// TwinCAT 3 PLC project PRG_MachineSystem
// Title: B_MachineSystem
// Company: RafalOS
// Author: Rafał Osajda
// ProjectVersion: 0.0.0.19
// ProgramVersion: 3.1.4024.0
// libraries:
//   B_Base, * (RafalOS)
//   B_Base_HMI_Connector, * (RafalOS)
//   B_HMIElements, * (RafalOS)
//   B_HMIManager, * (RafałOS)
//   B_IO, * (RafalOS)
//   B_MachineControl, * (RafalOS)
//   B_MachineControl_HMI_Connector, * (RafalOS)
//   B_StatesAndModes, * (RafalOS)
//   Tc2_Standard, * (Beckhoff Automation GmbH)
//   Tc2_System, * (Beckhoff Automation GmbH)
//   Tc3_Module, * (Beckhoff Automation GmbH)
// project tree:
//   GVLs/ GVL_MCSafety.TcGVL, GVL_RequeestChange.TcGVL, GVL_SystemVariable.TcGVL
//   / PlcTask.TcTTO
//   POUsCompilation/ Compilation.TcPOU
//   POUs/01_MachineDefaultConfiguration/ FB_MachineDefaultConfiguration.TcPOU
//   POUs/02_HMIDefaultConfiguration/ FB_DefaultHMIConfiguration.TcPOU
//   POUs/03_CreatingTempleteRecipe/ FB_DefaultTemplate.TcPOU
//   POUs/ PRG_ControlHMI.TcPOU, PRG_ControlHMIInit.TcPOU, PRG_SystemControlMachineInit.TcPOU, PRG_SystemControlMachineWork.TcPOU, ST_MainMenuButton.TcDUT, ST_PrepareDataModules.TcDUT

CONFIGURATION PRG_MachineSystem
    RESOURCE PLC ON TwinCAT3
        TASK PlcTask(INTERVAL := T#10ms, PRIORITY := 20);
        PROGRAM Compilation WITH PlcTask : Compilation;
        PROGRAM PRG_ControlHMI WITH PlcTask : PRG_ControlHMI;
        PROGRAM PRG_SystemControlMachineInit WITH PlcTask : PRG_SystemControlMachineInit;
        PROGRAM PRG_SystemControlMachineWork WITH PlcTask : PRG_SystemControlMachineWork;
        PROGRAM PRG_ControlHMIInit WITH PlcTask : PRG_ControlHMIInit;
    END_RESOURCE
END_CONFIGURATION

// ---- POUs/ST_MainMenuButton.TcDUT
TYPE ST_MainMenuButton :
STRUCT
	fbMMB0_MainScreen			: FB_HMIEButton;
	fbMMB1_Recipe				: FB_HMIEButton;
	fbMMB2_Parameters			: FB_HMIEButton;
	fbMMB3_Events				: FB_HMIEButton;
	fbMMB4_ModeChange			: FB_HMIEButton;
	fbMMB5_Statistics			: FB_HMIEButton;
	fbMMB6_StateDiagram			: FB_HMIEButton;
	fbMMB7_Settings				: FB_HMIEButton;

	fbMMB0_MainScreen_HMI_Connector		: FB_HMIEButton_HMI (itfBaseLoggerConnector := GVL_SystemVariable.fbLogger, itfButton := fbMMB0_MainScreen);
	fbMMB1_Recipe_HMI_Connector			: FB_HMIEButton_HMI (itfBaseLoggerConnector := GVL_SystemVariable.fbLogger, itfButton := fbMMB1_Recipe);
	fbMMB2_Parameters_HMI_Connector		: FB_HMIEButton_HMI (itfBaseLoggerConnector := GVL_SystemVariable.fbLogger, itfButton := fbMMB2_Parameters);
	fbMMB3_Events_HMI_Connector			: FB_HMIEButton_HMI (itfBaseLoggerConnector := GVL_SystemVariable.fbLogger, itfButton := fbMMB3_Events);
	fbMMB4_ModeChange_HMI_Connector		: FB_HMIEButton_HMI (itfBaseLoggerConnector := GVL_SystemVariable.fbLogger, itfButton := fbMMB4_ModeChange);
	fbMMB5_Statistics_HMI_Connector		: FB_HMIEButton_HMI (itfBaseLoggerConnector := GVL_SystemVariable.fbLogger, itfButton := fbMMB5_Statistics);
	fbMMB6_StateDiagram_HMI_Connector	: FB_HMIEButton_HMI (itfBaseLoggerConnector := GVL_SystemVariable.fbLogger, itfButton := fbMMB6_StateDiagram);
	fbMMB7_Settings_HMI_Connector		: FB_HMIEButton_HMI (itfBaseLoggerConnector := GVL_SystemVariable.fbLogger, itfButton := fbMMB7_Settings);
	
END_STRUCT
END_TYPE

// ---- POUs/ST_PrepareDataModules.TcDUT
TYPE ST_PrepareDataModules :
STRUCT
	fbPrepareDataModul_Empty			: FB_MCHMIPrepareDataForScreen;
	fbPrepareDataModul_00_01			: FB_MCHMIPrepareDataForScreen_00_01;
	fbPrepareDataModul_00_02			: FB_MCHMIPrepareDataForScreen_00_02;
	fbPrepareDataModul_00_03			: FB_MCHMIPrepareDataForScreen_00_03;
	fbPrepareDataModul_00_04			: FB_MCHMIPrepareDataForScreen_00_04;
	fbPrepareDataModul_00_05			: FB_MCHMIPrepareDataForScreen_00_05;
	fbPrepareDataModul_01_XX			: FB_MCHMIPrepareDataForScreen_01_XX;	//parametry
	fbPrepareDataModul_02_XX			: FB_MCHMIPrepareDataForScreen_02_XX;	//receptury
	fbPrepareDataModul_03_XX			: FB_MCHMIPrepareDataForScreen_03_XX;	//alarmy 
	fbPrepareDataModul_04_XX			: FB_MCHMIPrepareDataForScreen_04_XX;	//zmiana trybu
	fbPrepareDataModul_05_XX			: FB_MCHMIPrepareDataForScreen_05_XX;	//statystyki
	fbPrepareDataModul_06_XX			: FB_MCHMIPrepareDataForScreen_06_XX;	//diagram
	fbPrepareDataModul_07_XX			: FB_MCHMIPrepareDataForScreen_07_XX;	//ustawienia
END_STRUCT
END_TYPE

// ---- GVLs/GVL_MCSafety.TcGVL
{attribute 'qualified_only'}
VAR_GLOBAL
	flSS1				: FB_BaseFlag;
	flSTO				: FB_BaseFlag;
	
END_VAR

// ---- GVLs/GVL_RequeestChange.TcGVL
{attribute 'qualified_only'}
VAR_GLOBAL
//Przyciski zmaiany stanu	
//	fbprUndefined			: FB_RequestChanges;
	fbprAbort				: FB_MCRequiredChange;
  	fbprClear				: FB_MCRequiredChange;
   	fbprReset				: FB_MCRequiredChange;
   	fbprStart				: FB_MCRequiredChange;
   	fbprStop				: FB_MCRequiredChange;
   	fbprHold				: FB_MCRequiredChange;
   	fbprUnhold				: FB_MCRequiredChange;
   	fbprSuspend				: FB_MCRequiredChange;
   	fbprUnsuspend			: FB_MCRequiredChange;
  	fbprComplete			: FB_MCRequiredChange;
//przyciski zmiany trybu
//	fbprNiedozwolony		: FB_SITP_PolecenieZmianyTrybu (ePolecenie := E_SITP_PolecenieZmianyTrybu.brak);     
	fbprProduction			: FB_MCRequiredChange;
    fbprMaintenance			: FB_MCRequiredChange;
    fbprManual				: FB_MCRequiredChange;
    fbprWashing				: FB_MCRequiredChange;
    fbprDiagnostics			: FB_MCRequiredChange;
//    fbprUzytkownika2		: FB_RequestChanges;
//   fbprUzytkownika3		: FB_RequestChanges;
//    fbprUzytkownika4		: FB_RequestChanges;
//    fbprUzytkownika5		: FB_RequestChanges;

END_VAR

// ---- GVLs/GVL_SystemVariable.TcGVL
{attribute 'qualified_only'}
VAR_GLOBAL
	fbTime							: FB_BaseTime;
	fbLocation						: FB_BaseLocation;
	fbLogger						: FB_BaseLogger;
	stCommonData					: ST_BaseCommonData;
	
	(*	Element FB_MachineControl - sterowanie stanami i trybami pracy	*)
	fbSaMController					: FB_SaMController;
	
	(*	Główny element sterujący maszyną - logika pracy					*)
	fbMachineControl				: FB_MCMachineControl;
	
	(*	Zmienne zakończenia konfiguracji	*)
	bDefaultInitDone				: BOOL;
	bMachineInitDone				: BOOL;
	bControlHMIInit					: BOOL;
	
	(*	receptury	*)
	fbRecipe						: FB_BaseRecipe;
	
END_VAR

// ---- POUsCompilation/Compilation.TcPOU
PROGRAM Compilation
VAR
	fbMachineConfiguration	: FB_MachineDefaultConfiguration;
	fbHMIConfiguration		: FB_DefaultHMIConfiguration;
END_VAR

END_PROGRAM

// ---- POUs/01_MachineDefaultConfiguration/FB_MachineDefaultConfiguration.TcPOU
(*			
	RafalOS
	Rafał Osajda		10.11.2025		TC 4024.66
	Główny blok konfiguracyjny MachineControl
*)
FUNCTION_BLOCK FB_MachineDefaultConfiguration EXTENDS FB_Base IMPLEMENTS ITF_MCConfiguration
VAR

END_VAR

(*			
	RafalOS
	Rafał Osajda		26.11.2025		TC 4024.66
	Dodawanie szablonu receptury
*)
METHOD AddCreateTemplate : BOOL
VAR_INPUT
	itfMachineControl	: B_MachineControl.ITF_MCMachineControlConfigure;
END_VAR
//itfMachineControl.AddCreateTemplateFromConfiguration (fbCreateTemplate := );
END_METHOD

(*			
	RafalOS
	Rafał Osajda		13.11.2025		TC 4024.66
	Metoda przeznaczona do dodawania elementów do FB_MachineControl
*)
METHOD AddElements : BOOL
VAR_INPUT
	itfMachineControl	: B_MachineControl.ITF_MCMachineControlConfigure;
END_VAR
END_METHOD

(*			
	RafalOS
	Rafał Osajda		13.11.2025		TC 4024.66
	Podpięcie menadżera HMI
*)
METHOD AddHMIManager : BOOL
VAR_INPUT
	itfMachineControl	: B_MachineControl.ITF_MCMachineControlConfigure;
END_VAR
itfMachineControl.AddHMIManagerFromConfiguration (fbHMIManager := PRG_ControlHMI.fbHMIManager);
END_METHOD

(*			
	RafalOS
	Rafał Osajda		13.11.2025		TC 4024.66
	Dodanie samego siebie do systemu controli maszyny
*)
METHOD AddMachineCotrolToYourSelf : BOOL
VAR_INPUT
	itfMachineControl			: ITF_MCMachineControlConfigure;
END_VAR
itfMachineControl.AddMachineCotrolToYourSelfFromConfiguration ();
END_METHOD

(*			
	RafalOS
	Rafał Osajda		26.11.2025		TC 4024.66
	Dodanie obsługi receptur
*)
METHOD AddModulRecipe : BOOL
VAR_INPUT
	itfMachineControl	: B_MachineControl.ITF_MCMachineControlConfigure;
END_VAR
itfMachineControl.AddModulRecipeFromConfiguration (itfRecipe := GVL_SystemVariable.fbRecipe);
END_METHOD

(*			
	RafalOS
	Rafał Osajda		13.11.2025		TC 4024.66
	Dodanie modułu sterowania stanami i trybami do machinecontrol
*)
METHOD PUBLIC AddSaMCotrollerToMachineControl : BOOL
VAR_INPUT
	itfMachineControl			: ITF_MCMachineControlConfigure;
END_VAR
itfMachineControl.AddSaMCotrollerToMachineControlFromConfiguration (itfSaMController := GVL_SystemVariable.fbSaMController);
END_METHOD

METHOD AddSaMToTopElement
VAR_INPUT
	itfMachineControl	: B_MachineControl.ITF_MCMachineControlConfigure;
END_VAR
itfMachineControl.AddSaMToTopElementFromConfiguration (itfSaMController := GVL_SystemVariable.fbSaMController);
END_METHOD

(*			
	RafalOS
	Rafał Osajda		13.11.2025		TC 4024.66
	Zlinkowanie danych wspólnych do dodanych elementów
*)
METHOD LinkCommonDataToAddedElements : BOOL
VAR_INPUT
	itfMachineControl	: B_MachineControl.ITF_MCMachineControlConfigure;
END_VAR
itfMachineControl.LinkCommonDataToAddedElementsFromConfiguration (stCommonData := GVL_SystemVariable.stCommonData);
END_METHOD

(*			
	RafalOS
	Rafał Osajda		13.11.2025		TC 4024.66
	Dodanie głównego komunikatora pomiędzy topelementami do topelementów
*)
METHOD LinkMassangerToaddedTopElements : BOOL
VAR_INPUT
	itfMachineControl	: B_MachineControl.ITF_MCMachineControlConfigure;
END_VAR
itfMachineControl.LinkMassangerToaddedTopElementsFromConfiguration (
	fbCommunicator := GVL_SystemVariable.fbMachineControl.GetCommunicatorITF ()
);
END_METHOD

(*			
	RafalOS
	Rafał Osajda		14.11.2025		TC 4024.66
	Podpięcie przyciskow zmiany trybu i stanu
*)
METHOD LinkRequestButtonChange : BOOL
VAR_INPUT
	itfMachineControl	: B_MachineControl.ITF_MCMachineControlConfigure;
END_VAR
itfMachineControl.LinkRequestButtonStateChangeFromConfiguration (iNumberOfRequest := E_SaMCommandChangeState.Clear,		itfRequest := GVL_RequeestChange.fbprClear);
itfMachineControl.LinkRequestButtonStateChangeFromConfiguration (iNumberOfRequest := E_SaMCommandChangeState.Reset, 	itfRequest := GVL_RequeestChange.fbprReset);
itfMachineControl.LinkRequestButtonStateChangeFromConfiguration (iNumberOfRequest := E_SaMCommandChangeState.Start, 	itfRequest := GVL_RequeestChange.fbprStart);
itfMachineControl.LinkRequestButtonStateChangeFromConfiguration (iNumberOfRequest := E_SaMCommandChangeState.Stop, 		itfRequest := GVL_RequeestChange.fbprStop);
itfMachineControl.LinkRequestButtonStateChangeFromConfiguration (iNumberOfRequest := E_SaMCommandChangeState.Suspend, 	itfRequest := GVL_RequeestChange.fbprSuspend);
itfMachineControl.LinkRequestButtonStateChangeFromConfiguration (iNumberOfRequest := E_SaMCommandChangeState.Unsuspend, itfRequest := GVL_RequeestChange.fbprUnsuspend);
itfMachineControl.LinkRequestButtonStateChangeFromConfiguration (iNumberOfRequest := E_SaMCommandChangeState.Hold, 		itfRequest := GVL_RequeestChange.fbprHold);
itfMachineControl.LinkRequestButtonStateChangeFromConfiguration (iNumberOfRequest := E_SaMCommandChangeState.Unhold, 	itfRequest := GVL_RequeestChange.fbprUnhold);
itfMachineControl.LinkRequestButtonStateChangeFromConfiguration (iNumberOfRequest := E_SaMCommandChangeState.Complete, 	itfRequest := GVL_RequeestChange.fbprComplete);
itfMachineControl.LinkRequestButtonStateChangeFromConfiguration (iNumberOfRequest := E_SaMCommandChangeState.Abort,		itfRequest := GVL_RequeestChange.fbprAbort);

itfMachineControl.LinkRequestButtonModeChangeFromConfiguration (iNumberOfRequest := E_SaMCommandChangeMode.Production, 	itfRequest := GVL_RequeestChange.fbprProduction);
itfMachineControl.LinkRequestButtonModeChangeFromConfiguration (iNumberOfRequest := E_SaMCommandChangeMode.Maintenance,	itfRequest := GVL_RequeestChange.fbprMaintenance);
itfMachineControl.LinkRequestButtonModeChangeFromConfiguration (iNumberOfRequest := E_SaMCommandChangeMode.Manual, 		itfRequest := GVL_RequeestChange.fbprManual);
itfMachineControl.LinkRequestButtonModeChangeFromConfiguration (iNumberOfRequest := E_SaMCommandChangeMode.Washing,		itfRequest := GVL_RequeestChange.fbprWashing);
itfMachineControl.LinkRequestButtonModeChangeFromConfiguration (iNumberOfRequest := E_SaMCommandChangeMode.Diagnostisc,	itfRequest := GVL_RequeestChange.fbprDiagnostics);
END_METHOD

(*			
	RafalOS
	Rafał Osajda		13.11.2025		TC 4024.66
	Podłączenie wsyzstkich zmiennych pochodzących od Programu safety 
*)
METHOD LinkSafetyToaddedElements : BOOL
VAR_INPUT
	itfMachineControl	: B_MachineControl.ITF_MCMachineControlConfigure;
END_VAR
itfMachineControl.LinkSafetyToaddedElementsFromConfiguration (
	flSS1 := GVL_MCSafety.flSS1,
	flSTO := GVL_MCSafety.flSTO
);
END_METHOD

(*			
	RafalOS
	Rafał Osajda		13.11.2025		TC 4024.66
	Nadanie unikalnych kodów elementom w systemie
*)
METHOD SetCodeToAddedElements : BOOL
VAR_INPUT
	itfMachineControl	: B_MachineControl.ITF_MCMachineControlConfigure;
END_VAR
itfMachineControl.SetCodeToAddedElementsFromConfiguration ();
END_METHOD

(*			
	RafalOS
	Rafał Osajda		13.11.2025		TC 4024.66
	Uruchomienie lub wyłączenie obsługi HMI jak jest false fb obsługi nie jest dodawane do MachineControl
*)
METHOD SetEnableHMIService : BOOL
VAR_INPUT
	itfMachineControl	: B_MachineControl.ITF_MCMachineControlConfigure;
END_VAR
itfMachineControl.SetEnableHMIServiceFromConfiguration (bValue := TRUE);
END_METHOD

(*			
	RafalOS
	Rafał Osajda		13.11.2025		TC 4024.66
	Nadaje unikalne ID zgłoszeniom dodanym do elementów w sesyemie
*)
METHOD SetIDEventsToAddedElements : BOOL
VAR_INPUT
	itfMachineControl	: B_MachineControl.ITF_MCMachineControlConfigure;
END_VAR
itfMachineControl.SetIDEventsToAddedElementsFromConfiguration ();
END_METHOD

(*			
	RafalOS
	Rafał Osajda		13.11.2025		TC 4024.66
	Dodanie wszystkim elementom w systemie unikalnego ID
*)
METHOD SetIDToAddedElements : BOOL
VAR_INPUT
	itfMachineControl	: B_MachineControl.ITF_MCMachineControlConfigure;
END_VAR
itfMachineControl.SetIDToAddedElementsFromConfiguration ();
END_METHOD

(*			
	RafalOS
	Rafał Osajda		14.11.2025		TC 4024.66
	ustawienie trybu poczatkowego
*)
METHOD SetStartMode : BOOL
VAR_INPUT
	itfMachineControl	: B_MachineControl.ITF_MCMachineControlConfigure;
END_VAR
itfMachineControl.SetStartModeFromConfiguration (eStartMode := E_BaseMachineMode.Production);
END_METHOD

METHOD PUBLIC STARE_AddHMIToMachineControl : BOOL
VAR_INPUT
	itfMachineControl			: ITF_MCMachineControlConfigure;
END_VAR
//itfMachineControl.AddHMIManager (itfHMIManager := GVL_SystemVariable.fbHMIManager);
END_METHOD

METHOD PUBLIC STARE_AddTopElementToLogger : BOOL
VAR_INPUT
END_VAR
//GVL_SystemVariable.fbMachineControl.JoinTheLogger ();
END_METHOD

(*			
	RafalOS
	Rafał Osajda		29.10.2025		TC 4024.66
	Dodawanie TopElementu do systemu
*)
METHOD PUBLIC STARE_AddTopElementToMachineControl : BOOL
VAR_INPUT
	itfMachineControl			: ITF_MCMachineControlConfigure;
END_VAR
//THIS^.SetText (eLocation := E_BaseLocation.pl, wsDescription := "System");
//THIS^.SetText (eLocation := E_BaseLocation.en, wsDescription := "System");
//THIS^.SetText (eLocation := E_BaseLocation.de, wsDescription := "System");
//GVL_SystemVariable.fbMachineControl.SetName (stName := THIS^.GetTexts ());
//itfMachineControl.AddTopElementFromConfiguration (fbTopElement	:= GVL_SystemVariable.fbMachineControl);
END_METHOD

METHOD STARE_StateAndModes : BOOL
VAR_INPUT
	itfMachineControl			: ITF_MCMachineControlConfigure;
END_VAR
//itfMachineControl.AddRequestStateChange (iNumberOfRequest := E_SaMCommandChangeState.Clear,		itfRequest := GVL_RequeestChange.fbprClear);
//itfMachineControl.AddRequestStateChange (iNumberOfRequest := E_SaMCommandChangeState.Reset, 	itfRequest := GVL_RequeestChange.fbprReset);
//itfMachineControl.AddRequestStateChange (iNumberOfRequest := E_SaMCommandChangeState.Start, 	itfRequest := GVL_RequeestChange.fbprStart);
//itfMachineControl.AddRequestStateChange (iNumberOfRequest := E_SaMCommandChangeState.Stop, 		itfRequest := GVL_RequeestChange.fbprStop);
//itfMachineControl.AddRequestStateChange (iNumberOfRequest := E_SaMCommandChangeState.Suspend, 	itfRequest := GVL_RequeestChange.fbprSuspend);
//itfMachineControl.AddRequestStateChange (iNumberOfRequest := E_SaMCommandChangeState.Unsuspend, itfRequest := GVL_RequeestChange.fbprUnsuspend);
//itfMachineControl.AddRequestStateChange (iNumberOfRequest := E_SaMCommandChangeState.Hold, 		itfRequest := GVL_RequeestChange.fbprHold);
//itfMachineControl.AddRequestStateChange (iNumberOfRequest := E_SaMCommandChangeState.Unhold, 	itfRequest := GVL_RequeestChange.fbprUnhold);
//itfMachineControl.AddRequestStateChange (iNumberOfRequest := E_SaMCommandChangeState.Complete, 	itfRequest := GVL_RequeestChange.fbprComplete);
//itfMachineControl.AddRequestStateChange (iNumberOfRequest := E_SaMCommandChangeState.Abort,		itfRequest := GVL_RequeestChange.fbprAbort);
//
//itfMachineControl.AddRequestModeChange (iNumberOfRequest := E_SaMCommandChangeMode.Production, 	itfRequest := GVL_RequeestChange.fbprProduction);
//itfMachineControl.AddRequestModeChange (iNumberOfRequest := E_SaMCommandChangeMode.Maintenance,	itfRequest := GVL_RequeestChange.fbprMaintenance);
//itfMachineControl.AddRequestModeChange (iNumberOfRequest := E_SaMCommandChangeMode.Manual, 		itfRequest := GVL_RequeestChange.fbprManual);
//itfMachineControl.AddRequestModeChange (iNumberOfRequest := E_SaMCommandChangeMode.Washing,		itfRequest := GVL_RequeestChange.fbprWashing);
//itfMachineControl.AddRequestModeChange (iNumberOfRequest := E_SaMCommandChangeMode.Diagnostisc,	itfRequest := GVL_RequeestChange.fbprDiagnostics);
END_METHOD

END_FUNCTION_BLOCK

// ---- POUs/PRG_ControlHMI.TcPOU
(*			
	RafalOS
	Rafał Osajda		10.11.2025		TC 4024.66
	Program sterowanie HMI
*)
PROGRAM PRG_ControlHMI
VAR
	(*	Domyślna struktura danych dla HMI	*)
	stHMIData					: ST_HMIManager;
	(*	Główny element sterowania wyświetlaniem na HMI					*)
	fbHMIManager				: FB_HMIManager;
	(*	Domyślne przyciski menu głównego - Logika i łaczniki do HMI	*)
	stMainMenuButton			: ST_MainMenuButton;
	(*	Menu główne - Logika 	*)
	fbMainMenu					: FB_HMIEMenu;
	(*	Menu główne - Łącznik	*)
	fbMainMenu_HMI_Connector	: FB_HMIEMenu_HMI (itfBaseLoggerConnector := GVL_SystemVariable.fbLogger, itfMenu := fbMainMenu);
	(*	Łącznik do Machine Control	*)
	fbMachineControl_HMI_Connector		: FB_MCHMIMachineControl_HMI (itfBaseLoggerConnector := GVL_SystemVariable.fbLogger, itfMachineControlConnector := GVL_SystemVariable.fbMachineControl);
	(*	Moduły przygotowyania danych dla stron	*)
	stPrepareDataModules		: ST_PrepareDataModules;
	(*	Łącznik do receptur		*)
	fbRecipeModul_HMI_Connector	: FB_BaseRecipe_HMI (fbBaseRecipe := GVL_SystemVariable.fbRecipe);
END_VAR


	(*	Wywołanie metody sterowania HMI	*)

IF (GVL_Systemvariable.bDefaultInitDone AND
	GVL_Systemvariable.bMachineInitDone AND
	GVL_SystemVariable.bControlHMIInit AND
	GVL_SystemVariable.fbMachineControl.IsInitDone ()) THEN
	
	fbHMIManager ();
END_IF

END_PROGRAM

// ---- POUs/02_HMIDefaultConfiguration/FB_DefaultHMIConfiguration.TcPOU
(*			
	RafalOS
	Rafał Osajda		10.11.2025		TC 4024.66
	Główny blok konfigurujący HMI
*)
FUNCTION_BLOCK FB_DefaultHMIConfiguration EXTENDS FB_Base IMPLEMENTS ITF_HMIConfiguration
VAR
END_VAR

(*			
	RafalOS
	Rafał Osajda		07.12.2025		TC 4024.66
	Dodawanie elementów do systemmu wyświetlania
*)
METHOD AddElement
VAR_INPUT
	itfHMIManager	: B_HMI_Manager.ITF_HMIManagerConfigure;
END_VAR
END_METHOD

(*			
	RafalOS
	Rafał Osajda		20.11.2025		TC 4024.66
	Dodawanie rozszerzonego wyświetlania danych inna prezenacja danych niż domyślna lista
*)
METHOD AddExtendedDisplayToPrepScrModule : BOOL
VAR_INPUT
	itfHMIManager	: B_HMI_Manager.ITF_HMIManagerConfigure;
END_VAR
//przykład jak rozszerzać w progframie maszyny 
//itfHMIManager.AddExtendedDisplayToPrepScrModuleFromConfiguration (
//	itfModule 		:= PRG_ControlHMI.fbPrepareDataModul_02_XX,
//	itfExtension 	:= PRG_ControlHMI.fbxxxx
//);
END_METHOD

(*			
	RafalOS
	Rafał Osajda		19.11.2025		TC 4024.66
	Dodanie połączenia do MachineControl
*)
METHOD AddMachineControlConnector : BOOL
VAR_INPUT
	itfHMIManager	: B_HMI_Manager.ITF_HMIManagerConfigure;
END_VAR
itfHMIManager.AddMachineControlConnectorFromConfiguration (
	itfMachineControl := PRG_ControlHMI.fbMachineControl_HMI_Connector
);
END_METHOD

(*			
	RafalOS
	Rafał Osajda		14.11.2025		TC 4024.66
	Dodanie do systemu menu głównego 
*)
METHOD AddMainMenu : BOOL
VAR_INPUT
	itfHMIManager	: B_HMI_Manager.ITF_HMIManagerConfigure;
END_VAR
	(*	Utowrzenie menu głównego	*)
THIS^.SetText (eLocation := E_BaseLocation.pl, wsDescription := "Okno główne");
THIS^.SetText (eLocation := E_BaseLocation.en, wsDescription := "Main screen");
THIS^.SetText (eLocation := E_BaseLocation.de, wsDescription := "Hauptbildschirm");
PRG_ControlHMI.stMainMenuButton.fbMMB0_MainScreen.SetName (stName := THIS^.GetTexts ());
PRG_ControlHMI.fbMainMenu.AddButton (fbButton :=PRG_ControlHMI.stMainMenuButton.fbMMB0_MainScreen);
THIS^.SetText (eLocation := E_BaseLocation.pl, wsDescription := "Receptury");
THIS^.SetText (eLocation := E_BaseLocation.en, wsDescription := "Recipe");
THIS^.SetText (eLocation := E_BaseLocation.de, wsDescription := "Rezept");
PRG_ControlHMI.stMainMenuButton.fbMMB1_Recipe.SetName (stName := THIS^.GetTexts ());
PRG_ControlHMI.fbMainMenu.AddButton (fbButton :=PRG_ControlHMI.stMainMenuButton.fbMMB1_Recipe);
THIS^.SetText (eLocation := E_BaseLocation.pl, wsDescription := "Parametry");
THIS^.SetText (eLocation := E_BaseLocation.en, wsDescription := "Parameters");
THIS^.SetText (eLocation := E_BaseLocation.de, wsDescription := "Parameter");
PRG_ControlHMI.stMainMenuButton.fbMMB2_Parameters.SetName (stName := THIS^.GetTexts ());
PRG_ControlHMI.fbMainMenu.AddButton (fbButton :=PRG_ControlHMI.stMainMenuButton.fbMMB2_Parameters);
THIS^.SetText (eLocation := E_BaseLocation.pl, wsDescription := "Zdarzenia");
THIS^.SetText (eLocation := E_BaseLocation.en, wsDescription := "Events");
THIS^.SetText (eLocation := E_BaseLocation.de, wsDescription := "Veranstaltungen");
PRG_ControlHMI.stMainMenuButton.fbMMB3_Events.SetName (stName := THIS^.GetTexts ());
PRG_ControlHMI.fbMainMenu.AddButton (fbButton :=PRG_ControlHMI.stMainMenuButton.fbMMB3_Events);
THIS^.SetText (eLocation := E_BaseLocation.pl, wsDescription := "Zmiana trybu");
THIS^.SetText (eLocation := E_BaseLocation.en, wsDescription := "Mode change");
THIS^.SetText (eLocation := E_BaseLocation.de, wsDescription := "Modusänderung");
PRG_ControlHMI.stMainMenuButton.fbMMB4_ModeChange.SetName (stName := THIS^.GetTexts ());
PRG_ControlHMI.fbMainMenu.AddButton (fbButton :=PRG_ControlHMI.stMainMenuButton.fbMMB4_ModeChange);
THIS^.SetText (eLocation := E_BaseLocation.pl, wsDescription := "Statystyki");
THIS^.SetText (eLocation := E_BaseLocation.en, wsDescription := "Statistics");
THIS^.SetText (eLocation := E_BaseLocation.de, wsDescription := "Statistiken");
PRG_ControlHMI.stMainMenuButton.fbMMB5_Statistics.SetName (stName := THIS^.GetTexts ());
PRG_ControlHMI.fbMainMenu.AddButton (fbButton :=PRG_ControlHMI.stMainMenuButton.fbMMB5_Statistics);
THIS^.SetText (eLocation := E_BaseLocation.pl, wsDescription := "Diagram stanów");
THIS^.SetText (eLocation := E_BaseLocation.en, wsDescription := "State diagram");
THIS^.SetText (eLocation := E_BaseLocation.de, wsDescription := "Zustandsdiagramm");
PRG_ControlHMI.stMainMenuButton.fbMMB6_StateDiagram.SetName (stName := THIS^.GetTexts ());
PRG_ControlHMI.fbMainMenu.AddButton (fbButton :=PRG_ControlHMI.stMainMenuButton.fbMMB6_StateDiagram);
THIS^.SetText (eLocation := E_BaseLocation.pl, wsDescription := "Ustawienia");
THIS^.SetText (eLocation := E_BaseLocation.en, wsDescription := "Settings");
THIS^.SetText (eLocation := E_BaseLocation.de, wsDescription := "Einstellungen");
PRG_ControlHMI.stMainMenuButton.fbMMB7_Settings.SetName (stName := THIS^.GetTexts ());
PRG_ControlHMI.fbMainMenu.AddButton (fbButton :=PRG_ControlHMI.stMainMenuButton.fbMMB7_Settings);
//
PRG_ControlHMI.fbMainMenu_HMI_Connector.AddButton (fbButtonHMI := PRG_ControlHMI.stMainMenuButton.fbMMB0_MainScreen_HMI_Connector);
PRG_ControlHMI.fbMainMenu_HMI_Connector.AddButton (fbButtonHMI := PRG_ControlHMI.stMainMenuButton.fbMMB1_Recipe_HMI_Connector);
PRG_ControlHMI.fbMainMenu_HMI_Connector.AddButton (fbButtonHMI := PRG_ControlHMI.stMainMenuButton.fbMMB2_Parameters_HMI_Connector);
PRG_ControlHMI.fbMainMenu_HMI_Connector.AddButton (fbButtonHMI := PRG_ControlHMI.stMainMenuButton.fbMMB3_Events_HMI_Connector);
PRG_ControlHMI.fbMainMenu_HMI_Connector.AddButton (fbButtonHMI := PRG_ControlHMI.stMainMenuButton.fbMMB4_ModeChange_HMI_Connector);
PRG_ControlHMI.fbMainMenu_HMI_Connector.AddButton (fbButtonHMI := PRG_ControlHMI.stMainMenuButton.fbMMB5_Statistics_HMI_Connector);
PRG_ControlHMI.fbMainMenu_HMI_Connector.AddButton (fbButtonHMI := PRG_ControlHMI.stMainMenuButton.fbMMB6_StateDiagram_HMI_Connector);
PRG_ControlHMI.fbMainMenu_HMI_Connector.AddButton (fbButtonHMI := PRG_ControlHMI.stMainMenuButton.fbMMB7_Settings_HMI_Connector);

itfHMIManager.AddMainMenuFromConfiguration (
	fbMenu := PRG_ControlHMI.fbMainMenu,
	fbMenu_HMI := PRG_ControlHMI.fbMainMenu_HMI_Connector
);
END_METHOD

(*			
	RafalOS
	Rafał Osajda		19.11.2025		TC 4024.66
	Dodanie modułów do przygotowywania stron do wyświetlenia
*)
METHOD AddPrepareScreenModule : BOOL
VAR_INPUT
	itfHMIManager	: B_HMI_Manager.ITF_HMIManagerConfigure;
END_VAR
VAR
	iforScreen	: INT;
	iforMode	: INT;
END_VAR
	(*	Dodanie modułów do machine controil	*)
itfHMIManager.AddPrepareScreenModuleFromConfiguration (itfModule := PRG_ControlHMI.stPrepareDataModules.fbPrepareDataModul_Empty);
itfHMIManager.AddPrepareScreenModuleFromConfiguration (itfModule := PRG_ControlHMI.stPrepareDataModules.fbPrepareDataModul_00_01);
itfHMIManager.AddPrepareScreenModuleFromConfiguration (itfModule := PRG_ControlHMI.stPrepareDataModules.fbPrepareDataModul_00_02);
itfHMIManager.AddPrepareScreenModuleFromConfiguration (itfModule := PRG_ControlHMI.stPrepareDataModules.fbPrepareDataModul_00_03);
itfHMIManager.AddPrepareScreenModuleFromConfiguration (itfModule := PRG_ControlHMI.stPrepareDataModules.fbPrepareDataModul_00_04);
itfHMIManager.AddPrepareScreenModuleFromConfiguration (itfModule := PRG_ControlHMI.stPrepareDataModules.fbPrepareDataModul_00_05);
itfHMIManager.AddPrepareScreenModuleFromConfiguration (itfModule := PRG_ControlHMI.stPrepareDataModules.fbPrepareDataModul_01_XX);
itfHMIManager.AddPrepareScreenModuleFromConfiguration (itfModule := PRG_ControlHMI.stPrepareDataModules.fbPrepareDataModul_02_XX);
itfHMIManager.AddPrepareScreenModuleFromConfiguration (itfModule := PRG_ControlHMI.stPrepareDataModules.fbPrepareDataModul_03_XX);
itfHMIManager.AddPrepareScreenModuleFromConfiguration (itfModule := PRG_ControlHMI.stPrepareDataModules.fbPrepareDataModul_04_XX);
itfHMIManager.AddPrepareScreenModuleFromConfiguration (itfModule := PRG_ControlHMI.stPrepareDataModules.fbPrepareDataModul_05_XX);
itfHMIManager.AddPrepareScreenModuleFromConfiguration (itfModule := PRG_ControlHMI.stPrepareDataModules.fbPrepareDataModul_06_XX);
itfHMIManager.AddPrepareScreenModuleFromConfiguration (itfModule := PRG_ControlHMI.stPrepareDataModules.fbPrepareDataModul_07_XX);


	(*	Przypisanie do wszystkich pól pustego FB *)
FOR iforScreen := 0 TO GVL_HMIEConstans.MAX_NUMBER_OF_BUTTON_IN_MENU DO 
	FOR iforMode := 0 TO GVL_SaMConstans.NUMBER_OF_MODES DO 
		itfHMIManager.LinkPrepareScreenToArrayFromConfiguration (
			iScreen 	:= iforScreen, 
			iMode 		:= iforMode, 
			itfModule 	:= PRG_ControlHMI.stPrepareDataModules.fbPrepareDataModul_Empty
		);
	END_FOR
END_FOR

PRG_ControlHMI.stPrepareDataModules.fbPrepareDataModul_00_01.LinkMachineControlHMI (fbMachineControlHMI := PRG_ControlHMI.fbMachineControl_HMI_Connector);
PRG_ControlHMI.stPrepareDataModules.fbPrepareDataModul_00_02.LinkMachineControlHMI (fbMachineControlHMI := PRG_ControlHMI.fbMachineControl_HMI_Connector);
PRG_ControlHMI.stPrepareDataModules.fbPrepareDataModul_00_03.LinkMachineControlHMI (fbMachineControlHMI := PRG_ControlHMI.fbMachineControl_HMI_Connector);
PRG_ControlHMI.stPrepareDataModules.fbPrepareDataModul_00_04.LinkMachineControlHMI (fbMachineControlHMI := PRG_ControlHMI.fbMachineControl_HMI_Connector);
PRG_ControlHMI.stPrepareDataModules.fbPrepareDataModul_00_05.LinkMachineControlHMI (fbMachineControlHMI := PRG_ControlHMI.fbMachineControl_HMI_Connector);
PRG_ControlHMI.stPrepareDataModules.fbPrepareDataModul_01_XX.LinkMachineControlHMI (fbMachineControlHMI := PRG_ControlHMI.fbMachineControl_HMI_Connector);
PRG_ControlHMI.stPrepareDataModules.fbPrepareDataModul_02_XX.LinkMachineControlHMI (fbMachineControlHMI := PRG_ControlHMI.fbMachineControl_HMI_Connector);
PRG_ControlHMI.stPrepareDataModules.fbPrepareDataModul_03_XX.LinkMachineControlHMI (fbMachineControlHMI := PRG_ControlHMI.fbMachineControl_HMI_Connector);
PRG_ControlHMI.stPrepareDataModules.fbPrepareDataModul_04_XX.LinkMachineControlHMI (fbMachineControlHMI := PRG_ControlHMI.fbMachineControl_HMI_Connector);
PRG_ControlHMI.stPrepareDataModules.fbPrepareDataModul_05_XX.LinkMachineControlHMI (fbMachineControlHMI := PRG_ControlHMI.fbMachineControl_HMI_Connector);
PRG_ControlHMI.stPrepareDataModules.fbPrepareDataModul_06_XX.LinkMachineControlHMI (fbMachineControlHMI := PRG_ControlHMI.fbMachineControl_HMI_Connector);
PRG_ControlHMI.stPrepareDataModules.fbPrepareDataModul_07_XX.LinkMachineControlHMI (fbMachineControlHMI := PRG_ControlHMI.fbMachineControl_HMI_Connector);

	(*	Przypisanie modułów do aktywnych akien 	*)
itfHMIManager.LinkPrepareScreenToArrayFromConfiguration (iScreen := 0, iMode := 1, itfModule := PRG_ControlHMI.stPrepareDataModules.fbPrepareDataModul_00_01);
itfHMIManager.LinkPrepareScreenToArrayFromConfiguration (iScreen := 0, iMode := 2, itfModule := PRG_ControlHMI.stPrepareDataModules.fbPrepareDataModul_00_02);
itfHMIManager.LinkPrepareScreenToArrayFromConfiguration (iScreen := 0, iMode := 3, itfModule := PRG_ControlHMI.stPrepareDataModules.fbPrepareDataModul_00_03);
itfHMIManager.LinkPrepareScreenToArrayFromConfiguration (iScreen := 0, iMode := 4, itfModule := PRG_ControlHMI.stPrepareDataModules.fbPrepareDataModul_00_04);
itfHMIManager.LinkPrepareScreenToArrayFromConfiguration (iScreen := 0, iMode := 5, itfModule := PRG_ControlHMI.stPrepareDataModules.fbPrepareDataModul_00_05);

itfHMIManager.LinkPrepareScreenToArrayFromConfiguration (iScreen := 1, iMode := 1, itfModule := PRG_ControlHMI.stPrepareDataModules.fbPrepareDataModul_01_XX);
itfHMIManager.LinkPrepareScreenToArrayFromConfiguration (iScreen := 1, iMode := 2, itfModule := PRG_ControlHMI.stPrepareDataModules.fbPrepareDataModul_01_XX);
itfHMIManager.LinkPrepareScreenToArrayFromConfiguration (iScreen := 1, iMode := 3, itfModule := PRG_ControlHMI.stPrepareDataModules.fbPrepareDataModul_01_XX);
itfHMIManager.LinkPrepareScreenToArrayFromConfiguration (iScreen := 1, iMode := 4, itfModule := PRG_ControlHMI.stPrepareDataModules.fbPrepareDataModul_01_XX);
itfHMIManager.LinkPrepareScreenToArrayFromConfiguration (iScreen := 1, iMode := 5, itfModule := PRG_ControlHMI.stPrepareDataModules.fbPrepareDataModul_01_XX);

itfHMIManager.LinkPrepareScreenToArrayFromConfiguration (iScreen := 2, iMode := 1, itfModule := PRG_ControlHMI.stPrepareDataModules.fbPrepareDataModul_02_XX);
itfHMIManager.LinkPrepareScreenToArrayFromConfiguration (iScreen := 2, iMode := 2, itfModule := PRG_ControlHMI.stPrepareDataModules.fbPrepareDataModul_02_XX);
itfHMIManager.LinkPrepareScreenToArrayFromConfiguration (iScreen := 2, iMode := 3, itfModule := PRG_ControlHMI.stPrepareDataModules.fbPrepareDataModul_02_XX);
itfHMIManager.LinkPrepareScreenToArrayFromConfiguration (iScreen := 2, iMode := 4, itfModule := PRG_ControlHMI.stPrepareDataModules.fbPrepareDataModul_02_XX);
itfHMIManager.LinkPrepareScreenToArrayFromConfiguration (iScreen := 2, iMode := 5, itfModule := PRG_ControlHMI.stPrepareDataModules.fbPrepareDataModul_02_XX);

itfHMIManager.LinkPrepareScreenToArrayFromConfiguration (iScreen := 3, iMode := 1, itfModule := PRG_ControlHMI.stPrepareDataModules.fbPrepareDataModul_03_XX);
itfHMIManager.LinkPrepareScreenToArrayFromConfiguration (iScreen := 3, iMode := 2, itfModule := PRG_ControlHMI.stPrepareDataModules.fbPrepareDataModul_03_XX);
itfHMIManager.LinkPrepareScreenToArrayFromConfiguration (iScreen := 3, iMode := 3, itfModule := PRG_ControlHMI.stPrepareDataModules.fbPrepareDataModul_03_XX);
itfHMIManager.LinkPrepareScreenToArrayFromConfiguration (iScreen := 3, iMode := 4, itfModule := PRG_ControlHMI.stPrepareDataModules.fbPrepareDataModul_03_XX);
itfHMIManager.LinkPrepareScreenToArrayFromConfiguration (iScreen := 3, iMode := 5, itfModule := PRG_ControlHMI.stPrepareDataModules.fbPrepareDataModul_03_XX);

itfHMIManager.LinkPrepareScreenToArrayFromConfiguration (iScreen := 4, iMode := 1, itfModule := PRG_ControlHMI.stPrepareDataModules.fbPrepareDataModul_04_XX);
itfHMIManager.LinkPrepareScreenToArrayFromConfiguration (iScreen := 4, iMode := 2, itfModule := PRG_ControlHMI.stPrepareDataModules.fbPrepareDataModul_04_XX);
itfHMIManager.LinkPrepareScreenToArrayFromConfiguration (iScreen := 4, iMode := 3, itfModule := PRG_ControlHMI.stPrepareDataModules.fbPrepareDataModul_04_XX);
itfHMIManager.LinkPrepareScreenToArrayFromConfiguration (iScreen := 4, iMode := 4, itfModule := PRG_ControlHMI.stPrepareDataModules.fbPrepareDataModul_04_XX);
itfHMIManager.LinkPrepareScreenToArrayFromConfiguration (iScreen := 4, iMode := 5, itfModule := PRG_ControlHMI.stPrepareDataModules.fbPrepareDataModul_04_XX);

itfHMIManager.LinkPrepareScreenToArrayFromConfiguration (iScreen := 5, iMode := 1, itfModule := PRG_ControlHMI.stPrepareDataModules.fbPrepareDataModul_05_XX);
itfHMIManager.LinkPrepareScreenToArrayFromConfiguration (iScreen := 5, iMode := 2, itfModule := PRG_ControlHMI.stPrepareDataModules.fbPrepareDataModul_05_XX);
itfHMIManager.LinkPrepareScreenToArrayFromConfiguration (iScreen := 5, iMode := 3, itfModule := PRG_ControlHMI.stPrepareDataModules.fbPrepareDataModul_05_XX);
itfHMIManager.LinkPrepareScreenToArrayFromConfiguration (iScreen := 5, iMode := 4, itfModule := PRG_ControlHMI.stPrepareDataModules.fbPrepareDataModul_05_XX);
itfHMIManager.LinkPrepareScreenToArrayFromConfiguration (iScreen := 5, iMode := 5, itfModule := PRG_ControlHMI.stPrepareDataModules.fbPrepareDataModul_05_XX);

itfHMIManager.LinkPrepareScreenToArrayFromConfiguration (iScreen := 6, iMode := 1, itfModule := PRG_ControlHMI.stPrepareDataModules.fbPrepareDataModul_06_XX);
itfHMIManager.LinkPrepareScreenToArrayFromConfiguration (iScreen := 6, iMode := 2, itfModule := PRG_ControlHMI.stPrepareDataModules.fbPrepareDataModul_06_XX);
itfHMIManager.LinkPrepareScreenToArrayFromConfiguration (iScreen := 6, iMode := 3, itfModule := PRG_ControlHMI.stPrepareDataModules.fbPrepareDataModul_06_XX);
itfHMIManager.LinkPrepareScreenToArrayFromConfiguration (iScreen := 6, iMode := 4, itfModule := PRG_ControlHMI.stPrepareDataModules.fbPrepareDataModul_06_XX);
itfHMIManager.LinkPrepareScreenToArrayFromConfiguration (iScreen := 6, iMode := 5, itfModule := PRG_ControlHMI.stPrepareDataModules.fbPrepareDataModul_06_XX);

itfHMIManager.LinkPrepareScreenToArrayFromConfiguration (iScreen := 7, iMode := 1, itfModule := PRG_ControlHMI.stPrepareDataModules.fbPrepareDataModul_07_XX);
itfHMIManager.LinkPrepareScreenToArrayFromConfiguration (iScreen := 7, iMode := 2, itfModule := PRG_ControlHMI.stPrepareDataModules.fbPrepareDataModul_07_XX);
itfHMIManager.LinkPrepareScreenToArrayFromConfiguration (iScreen := 7, iMode := 3, itfModule := PRG_ControlHMI.stPrepareDataModules.fbPrepareDataModul_07_XX);
itfHMIManager.LinkPrepareScreenToArrayFromConfiguration (iScreen := 7, iMode := 4, itfModule := PRG_ControlHMI.stPrepareDataModules.fbPrepareDataModul_07_XX);
itfHMIManager.LinkPrepareScreenToArrayFromConfiguration (iScreen := 7, iMode := 5, itfModule := PRG_ControlHMI.stPrepareDataModules.fbPrepareDataModul_07_XX);
END_METHOD

(*			
	RafalOS
	Rafał Osajda		26.11.2025		TC 4024.66
	Podłaczenie modułu receptur
*)
METHOD AddRecipeModule : BOOL
VAR_INPUT
	itfHMIManager	: B_HMI_Manager.ITF_HMIManagerConfigure;
END_VAR
itfHMIManager.AddRecipeModuleFromConfiguration (fbRecipeModule := PRG_ControlHMI.fbRecipeModul_HMI_Connector);
END_METHOD

(*			
	RafalOS
	Rafał Osajda		18.11.2025		TC 4024.66
	Podłączenie głównej struktury danych dla domyślnych elementów 
*)
METHOD LinkHMIManagerData : BOOL
VAR_INPUT
	itfHMIManager	: B_HMI_Manager.ITF_HMIManagerConfigure;
END_VAR
itfHMIManager.LinkHMIManagerDataFromConfiguration (stData := PRG_ControlHMI.stHMIData);
END_METHOD

(*			
	RafalOS
	Rafał Osajda		16.12.2025		TC 4024.66
	Wywołanie linkowania zmiennych w topelemencie i jego dzieciach
*)
METHOD LinkMachineData : BOOL
VAR_INPUT
	itfHMIManager	: B_HMI_Manager.ITF_HMIManagerConfigure;
END_VAR
END_METHOD

(*			
	RafalOS
	Rafał Osajda		13.11.2025		TC 4024.66
	Podłączenie wsyzstkich zmiennych pochodzących od Programu safety 
*)
METHOD LinkSafetyToaddedElements : BOOL
VAR_INPUT
	itfHMIManager	: B_HMI_Manager.ITF_HMIManagerConfigure;
END_VAR
itfHMIManager.LinkSafetyToaddedElementsFromConfiguration (
	flSS1 := GVL_MCSafety.flSS1,
	flSTO := GVL_MCSafety.flSTO
);
END_METHOD

(*			
	RafalOS
	Rafał Osajda		18.11.2025		TC 4024.66
	Ustawia przycisk na aktywny  - pierwsze okno w wyświetlaniu wizualizacji
*)
METHOD SetButtonActive : BOOL
VAR_INPUT
	itfHMIManager	: B_HMI_Manager.ITF_HMIManagerConfigure;
END_VAR
itfHMIManager.SetButtonActiveFromConfiguration (iNumber := 0, bValue := TRUE);
END_METHOD

(*			
	RafalOS
	Rafał Osajda		18.11.2025		TC 4024.66
	Ustawia przyciski na wlaczone lub wylaczone - możliwośc naciśnięcia
*)
METHOD SetButtonsEnabled : BOOL
VAR_INPUT
	itfHMIManager	: B_HMI_Manager.ITF_HMIManagerConfigure;
END_VAR

VAR
	iI					: INT;
	iNumberofButtons	: INT;
END_VAR
iNumberofButtons := itfHMIManager.GetNumberOfAddedButtons ();
FOR iI := 0 TO iNumberofButtons DO
	itfHMIManager.SetButtonsEnabledFromConfiguration (iNumber := iI, bValue := TRUE);
END_FOR
END_METHOD

(*			
	RafalOS
	Rafał Osajda		18.11.2025		TC 4024.66
	Ustawia przyciski na widoczne lub nie widoczne
*)
METHOD SetButtonsVisible : BOOL
VAR_INPUT
	itfHMIManager	: B_HMI_Manager.ITF_HMIManagerConfigure;
END_VAR
VAR
	iI					: INT;
	iNumberofButtons	: INT;
END_VAR
iNumberofButtons := itfHMIManager.GetNumberOfAddedButtons ();
FOR iI := 0 TO iNumberofButtons DO
	itfHMIManager.SetButtonsEnabledFromConfiguration (iNumber := iI, bValue := TRUE);
END_FOR
END_METHOD

END_FUNCTION_BLOCK

// ---- POUs/PRG_SystemControlMachineInit.TcPOU
(*			
	RafalOS
	Rafał Osajda		25.10.2025		TC 4024.66
	Podpiecie zmiennych głównych do podzespołów 
*)
PROGRAM PRG_SystemControlMachineInit
VAR
	(*	Konfiguracja MachineControl	*)
	fbDefaultMachineConfiguration	: FB_MachineDefaultConfiguration;
	fbMachineConfigure				: FB_MCMachineConfigure;
	
END_VAR

IF (NOT GVL_SystemVariable.bDefaultInitDone AND 
	NOT GVL_SystemVariable.bMachineInitDone) THEN

	GVL_SystemVariable.stCommonData.itfTime := GVL_SystemVariable.fbTime;
	GVL_SystemVariable.stCommonData.itfLocaciotn := GVL_SystemVariable.fbLocation;
	GVL_SystemVariable.stCommonData.itfLogger := GVL_SystemVariable.fbLogger;

		(*	Podpięcie podstawowej konfiguracji	*)
	fbMachineConfigure.AddConfiguration (fbConfigure := fbDefaultMachineConfiguration);
	GVL_SystemVariable.fbMachineControl.AddModulConfigure (fbMachineConfigure := fbMachineConfigure);
		(*	Podpięcie danych do leogera 	*)
	GVL_SystemVariable.fbLogger.LinkCommonData (stCommonData := GVL_SystemVariable.stCommonData);
		(*	Podpięcie danych do receptur	*)
	GVL_SystemVariable.fbRecipe.LinkCommonData (stCommonData := GVL_SystemVariable.stCommonData);
		(* Pobranie ilosci szablonów jak nei ma żadnego szablonu to tworzymy *)
	

(*	
	(*	Linkowanie zmiennych z modułami	*)
	GVL_SystemVariable.fbLogger.LinkCommonData (stCommonData := GVL_SystemVariable.stCommonData);
	GVL_SystemVariable.fbMachineControl.LinkCommonData (stCommonData := GVL_SystemVariable.stCommonData);
	(*	Podpięcie zmiennych Safety		*)
	GVL_SystemVariable.fbMachineControl.LinkSS1 (fbSS1 := GVL_MCSafety.flSS1);
	GVL_SystemVariable.fbMachineControl.LinkSTO (fbSTO := GVL_MCSafety.flSTO);
	(*	Podpięcie zarządzania stanami i trybami pracy	*)
	GVL_SystemVariable.fbMachineControl.AddModulSaM (fbSaMController := GVL_SystemVariable.fbSaMController);
	
	GVL_SystemVariable.fbHMIManager.LinkCommonData (stCommonData := GVL_SystemVariable.stCommonData);
	(*	Podpięcie zmiennych Safety		*)
	GVL_SystemVariable.fbHMIManager.LinkSS1 (fbSS1 := GVL_MCSafety.flSS1);
	GVL_SystemVariable.fbHMIManager.LinkSTO (fbSTO := GVL_MCSafety.flSTO);
	
	
*)	
	GVL_SystemVariable.bDefaultInitDone	:= TRUE;
END_IF

END_PROGRAM

// ---- POUs/PRG_SystemControlMachineWork.TcPOU
PROGRAM PRG_SystemControlMachineWork
VAR
	bFirstCycle		: BOOL;
END_VAR

IF (GVL_SystemVariable.bDefaultInitDone AND
	GVL_SystemVariable.bMachineInitDone) THEN
	;
	(*	Wywołanie obsługi Logera	*)
	GVL_SystemVariable.fbLogger ();
	(*	Wywołanie pracy maszyny		*)
	GVL_SystemVariable.fbMachineControl ();
END_IF

END_PROGRAM

// ---- POUs/PRG_ControlHMIInit.TcPOU
PROGRAM PRG_ControlHMIInit
VAR
	(*	Konfiguracja HMIManager		*)
	fbDedaultHMIConfiguration		: FB_DefaultHMIConfiguration;
	fbHMIConfigure					: FB_HMIConfigure;
	
END_VAR

IF (NOT GVL_SystemVariable.bControlHMIInit) THEN
	GVL_SystemVariable.bControlHMIInit := TRUE;
		(*	Konfiguracjia systemu HMI	*)
	fbHMIConfigure.AddConfiguration (fbConfigure := fbDedaultHMIConfiguration);
	PRG_ControlHMI.fbHMIManager.AddModulConfigure (fbHMIConfigure := fbHMIConfigure);
	PRG_ControlHMI.fbRecipeModul_HMI_Connector.LinkCommonData (stCommonData := GVL_SystemVariable.stCommonData);
END_IF

END_PROGRAM

// ---- POUs/03_CreatingTempleteRecipe/FB_DefaultTemplate.TcPOU
FUNCTION_BLOCK FB_DefaultTemplate EXTENDS FB_Base IMPLEMENTS ITF_BaseCreateTemplateOfRecipe
VAR
END_VAR

METHOD CreateTamplateOfRecipe : BOOL
VAR_INPUT
	(*interfejs do obsługi receptur*)
	itfRecipe	: B_Base.ITF_BaseCreatingTemplateMethod;
END_VAR
(*	Metody tworzące szablon receptury 
	- dodanie nazwy i utworzenie szablonu 
	- dodawanie składników
*)
END_METHOD

END_FUNCTION_BLOCK
